PROGRAM PreInitialise
VAR
	iLoop  : INT := 0;
	bStartStep1 : BOOL := TRUE;
	tStartStep2 : TON;
	bStartStep2 : BOOL := FALSE;	
	tStartStep3 : TON;
	bStartStep3 : BOOL := FALSE;
	tStartStep4 : TON;
	bStartStep4 : BOOL := FALSE;
	
	stMLVIO : ST_TCMultiLevel_VIO;
	iLevel:Int:=1;
	noOfLevel: INT;
END_VAR

iTCColumnID		:= F_GetColumnID(eColumnID:=COLUMN_NAME);
F_GetModuleID(eColumnID:=COLUMN_NAME);


tStartStep2(IN:=bStartStep2, PT:=T#1S);
tStartStep3(IN:=bStartStep3, PT:=T#5S); 
tStartStep4(IN:=bStartStep4, PT:=T#1S);

IF bStartStep1 THEN
	bStartStep1 := FALSE;
	bStartStep2 := TRUE; //Proceed to step-2
	bStartStep3 := FALSE;
	bStartStep4 := FALSE;
	RETURN;
END_IF

IF tStartStep2.Q THEN
	
	Logging.fbDebugLog.M_nLogger(iLogLevel:= Logging.fbDebugLog.P_iLogVerbosity, sSource:= '', sMessage:= '                                                  ');
	Logging.fbDebugLog.M_nLogger(iLogLevel:= Logging.fbDebugLog.P_iLogVerbosity, sSource:= '', sMessage:= '                                                  ');
	Logging.fbDebugLog.M_nLogger(iLogLevel:= Logging.fbDebugLog.P_iLogVerbosity, sSource:= '', sMessage:= '==================================================');
	Logging.fbDebugLog.M_nLogger(iLogLevel:= Logging.fbDebugLog.P_iLogVerbosity, sSource:= '', sMessage:= 'AEM Singapore Pte Ltd. All rights reserved.       ');
	Logging.fbDebugLog.M_nLogger(iLogLevel:= Logging.fbDebugLog.P_iLogVerbosity, sSource:= '', sMessage:= '==================================================');
	Logging.fbDebugLog.M_nLogger(iLogLevel:= Logging.fbDebugLog.P_iLogVerbosity, sSource:= '', sMessage:= CONCAT(CONCAT('PLC TC v', stLibVersion_TC.sVersion), ' started'));
	Logging.fbDebugLog.M_nLogger(iLogLevel:= Logging.fbDebugLog.P_iLogVerbosity, sSource:= '', sMessage:= '                                                  ');	
	bGetAMSNetID:= TRUE;
	bStartStep1 := FALSE;
	bStartStep2 := FALSE; 
	bStartStep3 := TRUE; //Proceed to step-3
	bStartStep4 := FALSE;
	
	IF NOT bProductionMode THEN
		bEnableManualCommandTest1		:= TRUE;
		bEnableManualCommandTest2		:= TRUE;
		//IsNetIDReadOK					:= TRUE;
		//bDebugCart						:= FALSE;
	
	END_IF
	
	FOR iLevel:=1 TO NO_OF_LEVEL DO 
		GVL_EAP.stEAP.stTBOT_TC_EAP[iLevel].bAntiCollisionTriggered		:=TRUE;
		GVL_EAP.stEAP.stTBOT_TC_EAP[iLevel].bTCCellACPwrOff				:=FALSE;
		
		stMLVIO:=arrTCMultiLevel[iLevel].fbTCMultiLevelSeq.P_stTCMultiLevelVIO; //get method 
		
		
		//Lock back door if closed.
		IF stMLVIO.ipTCCellDoorOpenCloseStatus THEN
			stMLVIO.opCellDoorClosed 						:= TRUE;
		END_IF
		
		//Lock Front door if closed.
		IF bDebugCart THEN
			IF stMLVIO.ipTCCellTbotSideDoorOpenCloseStatus01 AND stMLVIO.ipTCCellTbotSideDoorOpenCloseStatus02 THEN
				stMLVIO.opCellTBOtSideDoorClosed1 		:= TRUE;
				stMLVIO.opCellTBOtSideDoorClosed2 		:= TRUE;
			END_IF
		END_IF
		
		stMLVIO.opAPAirSupplySol 							:= TRUE; //turn on all levels' AP 10bar 
		stMLVIO.opTesterDrawerAirSupplySol					:= TRUE; //turn on all levels' tester 6bar
		
		arrTCMultiLevel[iLevel].fbTCMultiLevelSeq.P_stTCMultiLevelVIO := stMLVIO; //set method
	END_FOR
	
	RETURN;
END_IF

IF tStartStep3.Q THEN
	bStartStep1 := FALSE;
	bStartStep2 := FALSE; 
	bStartStep3 := FALSE;
	bStartStep4 := TRUE;
	RETURN;
END_IF

IF tStartStep4.Q THEN
	//bPlcRunning := TRUE;
	
	bStartStep1 := FALSE;
	bStartStep2 := FALSE; 
	bStartStep3 := FALSE;
	bStartStep4 := FALSE;
	RETURN;
END_IF

END_PROGRAM

(* stored: Version 1.1.0.1, ProductVersion 3.1.4022.18
   POU PreInitialise: Id {1b25484a-6211-4e41-8f0e-ef1661458f4a}, SpecialFunc None *)
